TYPE
  (* Version 1.0, 2023-04-05, Tim Hesse *)
  ROS2_action_msgs__msg__GoalStatusArray : STRUCT
    status_list : ARRAY [0..15] OF ROS2_action_msgs__msg__GoalStatus;
  END_STRUCT;
END_TYPE
